// TwinCAT 3 PLC project PLC
// ProgramVersion: 3.1.4023.0
// libraries:
//   Tc2_Standard, * (Beckhoff Automation GmbH)
//   Tc2_System, * (Beckhoff Automation GmbH)
//   Tc3_Module, * (Beckhoff Automation GmbH)
//   VisuDialogs, * (System)
//   VisuSymbols,3.5.10.0,System
// project tree:
//   / GlobalTextList.TcGTLO, PlcTask.TcTTO, Visualization Manager.TcVMO (not stored)
//   POUs/ FB_Blinker.TcPOU, MAIN.TcPOU, pCounter.TcPOU
//   VISUs/ P03_Common.TcVIS, P00_Main.TcVIS, P02_Measurement.TcVIS, P01_Swtich_Lamp.TcVIS, P04_Table.TcVIS, TextList.TcTLO, W01_PopupScreen.TcVIS

CONFIGURATION PLC
    RESOURCE PLC ON TwinCAT3
        TASK PlcTask(INTERVAL := T#10ms, PRIORITY := 20);
        PROGRAM MAIN WITH PlcTask : MAIN;
    END_RESOURCE
END_CONFIGURATION

// ---- POUs/MAIN.TcPOU
PROGRAM MAIN
VAR 	
	bHmi_LAMP1  : BOOL;
	bHmi_LAMP2 : BOOL;
	bHmi_LAMP3  : BOOL;
	bHmi_LAMP4  : BOOL;
	
//	bOut_LAMP1  AT %Q*: BOOL;
//	bOut_LAMP2  AT %Q*: BOOL;
//	bOut_LAMP3  AT %Q*: BOOL;
//	bOut_LAMP4  AT %Q*: BOOL;
	
	bHmi_Swtic1 : BOOL;
	bHmi_Swtic2 : BOOL;
	bHmi_Swtic3 : BOOL;
	bHmi_Swtic4 : BOOL;
	
//	bIn_Swtic1 AT %I*: BOOL;
//	bIn_Swtic2 AT %I*: BOOL;
//	bIn_Swtic3 AT %I*: BOOL;
//	bIn_Swtic4 AT %I*: BOOL;
	
	iIN_VOLUME AT %I*: INT:=1000;
	
	//bIN_SW2 AT %I*: BOOL;
	fbBlinker: FB_Blinker;
	fbCTU: CTU;
	
	//HMI  BarDisplay
	iValueBarDisplay:INT;
	tTimer:TON;
	bDirection:BOOL;
	bValuePotentialMeter:INT;
	
	//Bar Graph
	lrSin:LREAL;
	aryLrSin:ARRAY[0..200] OF LREAL;
	tTimer2:TON;
	i:INT;
	
	//check Box
	bCheckBox:ARRAY[0..4] OF BOOL;
	bCheckBox1:BOOL;
	bCheckBox2:BOOL;
	bCheckBox3:BOOL;
	bCheckBox4:BOOL;
	bCheckBox5:BOOL;
	plsCheckBox1:R_trig;
	plsCheckBox2:R_trig;
	plsCheckBox3:R_trig;
	plsCheckBox4:R_trig;
	plsCheckBox5:R_trig;
	sOutput2:STRING;
	//Combbox and Radio Buttons
	iCombINdex:INT;
	sOutput:STRING;
	
    //Table 
	aryLrSin1:ARRAY[0..4,0..20] OF DINT;
	tTimer3:TON;
END_VAR

//bOUT_LAMP1:=bIN_SW1;
//iOUT_METER:=iIN_VOLUME;
//bOUT_LAMP3:= bIN_SW1 AND bIN_SW2;

//pCounter();

fbBlinker
(
//	bStart:=TRUE,
	bStart:=bHmi_Swtic1,
	tTime:=INT_TO_TIME(iIN_VOLUME),
	//bOutPut=>
);

fbCTU(
	CU:= fbBlinker.bOutPut, 
	RESET:= fbCTU.Q, 
	PV:= 4, 
	//Q=> , 
	//CV=> 
);

CASE fbCTU.CV OF 
	1: 
	bHmi_LAMP1:=TRUE;
	bHmi_LAMP2:=FALSE;
	bHmi_LAMP3:=FALSE;
	bHmi_LAMP4:=FALSE;
	2: 
	bHmi_LAMP1:=FALSE;
	bHmi_LAMP2:=TRUE;
	bHmi_LAMP3:=FALSE;
	bHmi_LAMP4:=FALSE;
	3: 
	bHmi_LAMP1:=FALSE;
	bHmi_LAMP2:=FALSE;
	bHmi_LAMP3:=TRUE;
	bHmi_LAMP4:=FALSE;
	4: 
	bHmi_LAMP1:=FALSE;
	bHmi_LAMP2:=FALSE;
	bHmi_LAMP3:=FALSE;
	bHmi_LAMP4:=TRUE;

END_CASE

//Hmi BarDisplay
tTimer(IN:=bHmi_Swtic2,PT:=T#10MS);
IF tTimer.Q THEN
	tTimer(IN:=FALSE);
	IF iValueBarDisplay = 1000 THEN
		bDirection:=TRUE;
	ELSIF iValueBarDisplay = 0 THEN
		bDirection:=FALSE;	
	END_IF
	
	IF bDirection THEN
		iValueBarDisplay:=iValueBarDisplay-1;
	ELSE
		iValueBarDisplay:=iValueBarDisplay+1;
	END_IF
END_IF

//HMI Bar Graph
lrSin:=SIN(TO_REAL(iValueBarDisplay)/1000);
tTimer2(IN:=bHmi_Swtic3,PT:=T#100MS);
IF tTimer2.Q THEN
	tTimer2(IN:=FALSE);
	FOR i:= 200 TO 1 BY -1 DO 
		aryLrSin[i]:=aryLrSin[i-1];
	END_FOR
	aryLrSin[0]:=LrSin;
END_IF
//CheckBox
plsCheckBox1(CLK:=bCheckBox1);
plsCheckBox2(CLK:=bCheckBox2);
plsCheckBox3(CLK:=bCheckBox3);
plsCheckBox4(CLK:=bCheckBox4);
plsCheckBox5(CLK:=bCheckBox5);
IF plsCheckBox1.Q THEN
	sOutput2:='Opton1';
	bCheckBox2:=FALSE;	
	bCheckBox3:=FALSE;	
	bCheckBox4:=FALSE;	
	bCheckBox5:=FALSE;	
ELSIF plsCheckBox2.Q THEN
	sOutput2:='Opton2';
	bCheckBox1:=FALSE;	
	bCheckBox3:=FALSE;	
	bCheckBox4:=FALSE;	
	bCheckBox5:=FALSE;	
ELSIF plsCheckBox3.Q THEN
	sOutput2:='Opton3';
	bCheckBox1:=FALSE;	
	bCheckBox2:=FALSE;	
	bCheckBox4:=FALSE;	
	bCheckBox5:=FALSE;		
ELSIF plsCheckBox4.Q THEN
	sOutput2:='Opton4';
	bCheckBox1:=FALSE;	
	bCheckBox2:=FALSE;	
	bCheckBox3:=FALSE;	
	bCheckBox5:=FALSE;	
ELSIF plsCheckBox5.Q THEN
	sOutput2:='Opton5';
	bCheckBox1:=FALSE;	
	bCheckBox2:=FALSE;	
	bCheckBox3:=FALSE;	
	bCheckBox4:=FALSE;	
END_IF
//CombBox
CASE iCombINdex OF
0:
 sOutput:='Opton1';
1:
 sOutput:='Opton2';
2:
 sOutput:='Opton3';
3:
 sOutput:='Opton4';
ELSE
 sOutput:='Error';
END_CASE
//Table
tTimer3(IN:=bHmi_Swtic4,PT:=T#1000MS);
IF tTimer3.Q THEN
	tTimer3(IN:=FALSE);
	FOR i:= 20 TO 1 BY -1 DO 
		aryLrSin1[0,i]:=aryLrSin1[0,i-1];
		aryLrSin1[1,i]:=aryLrSin1[1,i-1];
		aryLrSin1[2,i]:=aryLrSin1[2,i-1];
		aryLrSin1[3,i]:=aryLrSin1[3,i-1];
		aryLrSin1[4,i]:=aryLrSin1[4,i-1];
	END_FOR
	aryLrSin1[0,0]:=TO_DINT(LrSin*10000);
	aryLrSin1[1,0]:=TO_DINT(-LrSin*10000);
	aryLrSin1[2,0]:=TO_DINT((LrSin+1)*10000);
	aryLrSin1[3,0]:=TO_DINT((LrSin-1)*10000);
	aryLrSin1[4,0]:=TO_DINT((LrSin*2)*10000);
END_IF

END_PROGRAM

// ---- POUs/FB_Blinker.TcPOU
FUNCTION_BLOCK FB_Blinker
VAR_INPUT
	bStart: BOOL;
	tTime: TIME;
END_VAR
VAR_OUTPUT
	bOutPut: BOOL;
END_VAR
VAR
	T1: TON;
	T2: TON;
END_VAR

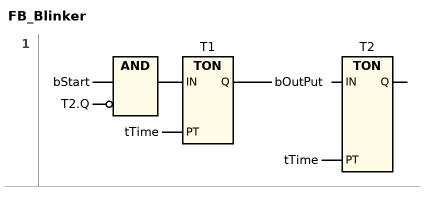
// NETWORK 1
T1(IN := bStart AND NOT T2.Q, PT := tTime); // TON
bOutPut := T1.Q;
T2(IN := T1.Q, PT := tTime); // TON

END_FUNCTION_BLOCK

// ---- POUs/pCounter.TcPOU
PROGRAM pCounter
VAR
	fbCTU: CTU;
	bSW1 AT %I*: BOOL;
	bSW2 AT %I*: BOOL;
	CurrentValue: WORD;
	bLED1 AT %Q*: BOOL;
END_VAR

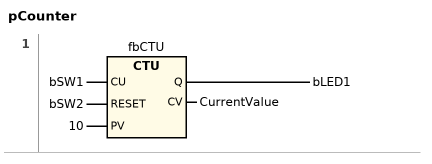
// NETWORK 1
fbCTU(CU := bSW1, RESET := bSW2, PV := 10, CV => CurrentValue); // CTU
bLED1 := fbCTU.Q;

END_PROGRAM

// ---- GlobalTextList.TcGTLO
TEXTLIST GlobalTextList
  646 = '%d'
  394 = '%s'
  322 = 'aryLrSiin1[1]'
  243 = 'aryLrSin1[0,INDEX]'
  253 = 'aryLrSin1[0]'
  589 = 'aryLrSin1[1,INDEX]'
  141 = 'aryLrSin1[1]'
  425 = 'aryLrSin1[2,INDEX]'
  682 = 'aryLrSin1[2]'
  644 = 'aryLrSin1[3,INDEX]'
  914 = 'aryLrSin1[3]'
  670 = 'aryLrSin1[4,INDEX]'
  300 = 'aryLrSin1[4]'
  706 = 'aryLrSin1[X]'
  594 = 'Bar_Switch_2'
  122 = 'Chart_Switch_3'
  446 = 'Check Box'
  607 = 'Check Box1'
  567 = 'Checkbox'
  756 = 'CheckBox'
  353 = 'Checkbox1'
  536 = 'Checkbox2'
  535 = 'Checkbox3'
  854 = 'Close Screen'
  739 = 'Close Window'
  413 = 'Common'
  320 = 'GroupBox'
  554 = 'Here PopUp\u3000'
  537 = 'Here PopUp\u3000TEXT\u3000'
  943 = 'Japanese'
  485 = 'Lamp_1' | JP: 'ランプ１'
  549 = 'Lamp_2' | JP: 'ランプ２'
  964 = 'Lamp_3' | JP: 'ランプ３'
  83 = 'Lamp_4' | JP: 'ランプ４'
  254 = 'Lamp_Switch_1'
  906 = 'Measument'
  348 = 'Measurement'
  331 = 'OpenPopup'
  733 = 'Option1'
  643 = 'Option14'
  808 = 'Option2'
  403 = 'Option3'
  186 = 'Option4'
  115 = 'Option5'
  754 = 'PopUp Window'
  588 = 'Switch 1'
  163 = 'Switch 2'
  482 = 'Switch 3'
  888 = 'Switch 4'
  357 = 'Switch Time' | JP: 'スイッチ時間'
  496 = 'Switch Time Act' | JP: '実時間'
  905 = 'Switch_1' | JP: 'スイッチ１'
  363 = 'Switch_2' | JP: 'スイッチ２'
  119 = 'Switch_3' | JP: 'スイッチ３'
  130 = 'Switch_4' | JP: 'スイッチ４'
  404 = 'swtich Lamp'
  929 = 'Swtich Time'
  542 = 'Table'
  559 = 'Table_Switch_4'
END_TEXTLIST

// ---- VISUs/P03_Common.TcVIS
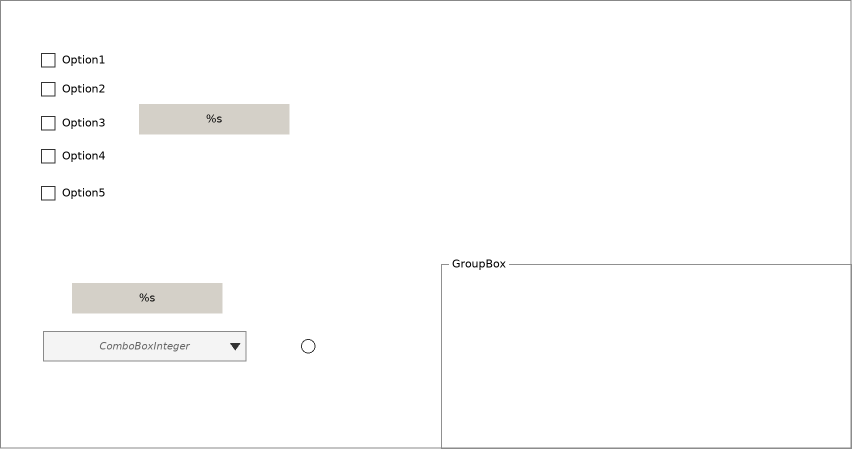
VISUALIZATION P03_Common  // 852x449
    Checkbox (39,45 150x30), "Option1", variable: Main.bCheckBox1
    Checkbox (39,74 150x30), "Option2", variable: Main.bCheckBox2
    Checkbox (39,108 150x30), "Option3", variable: Main.bCheckBox3
    Checkbox (39,141 150x30), "Option4", variable: Main.bCheckBox4
    Checkbox (39,178 150x30), "Option5", variable: Main.bCheckBox5
    Textfield (139,104 150x30), "%s", text variable: Main.sOutput2
    ComboBoxInteger (43,331 203x30), variable: Main.iCombINdex, text list: 'TextList'
    RadioButton (299,271 150x150), variable: Main.iCombINdex
        Areas[0]: Text=Option1
        Areas[1]: Text=Option2
        Areas[2]: Text=Option3
        Areas[3]: Text=Option4
        Areas[4]: Text=Option5
    Textfield (72,283 150x30), "%s", text variable: Main.sOutput
    GroupBox (441,256 411x193), "GroupBox"
END_VISUALIZATION

// ---- VISUs/P00_Main.TcVIS
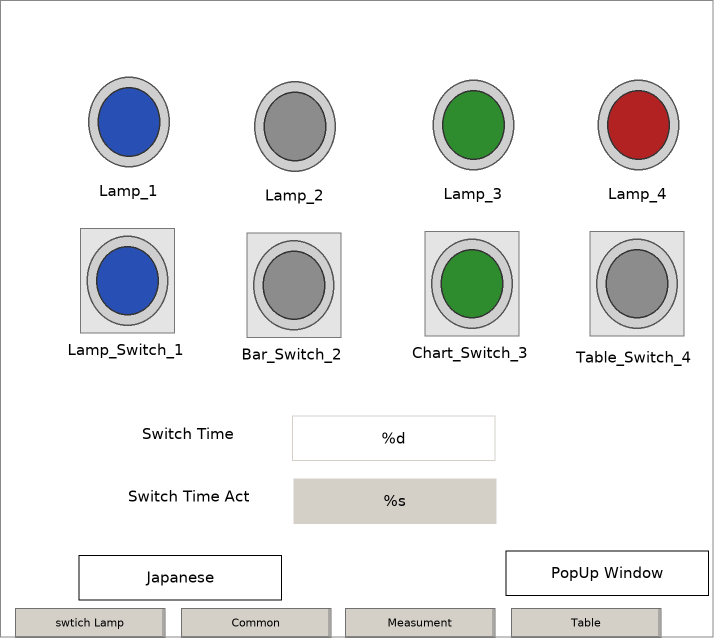
VISUALIZATION P00_Main  // 714x638
    Button (15,608 150x30), "swtich Lamp"
        OnMouseDown: FrameSelectionChange Selection=SelectedFrame=647e187a-0755-4409-bbed-ce6851db0410, GlobSel=AssignType=Directly, SelType=Locally
    Frame (29,26 685x574)
        shows P01_Swtich_Lamp()
        shows P02_Measurement()
        shows P03_Common()
        shows P04_Table()
    Button (181,608 150x30), "Common"
        OnMouseDown: FrameSelectionChange Selection=SelectedFrame=647e187a-0755-4409-bbed-ce6851db0410, Selection=2, GlobSel=AssignType=Directly, SelType=Locally
    Button (345,608 150x30), "Measument"
        OnMouseDown: FrameSelectionChange Selection=SelectedFrame=647e187a-0755-4409-bbed-ce6851db0410, Selection=1, GlobSel=AssignType=Directly, SelType=Locally
    Button (511,608 150x30), "Table"
        OnMouseDown: FrameSelectionChange Selection=SelectedFrame=647e187a-0755-4409-bbed-ce6851db0410, Selection=3, GlobSel=AssignType=Directly, SelType=Locally
END_VISUALIZATION

// ---- VISUs/P02_Measurement.TcVIS
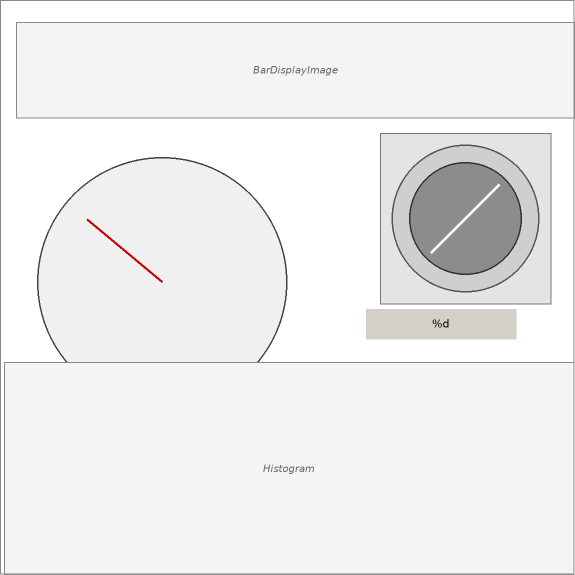
VISUALIZATION P02_Measurement  // 575x575
    BarDisplayImage (16,22 559x96), value: Main.iValueBarDisplay, style: BarDisplayImage-Gray, scale format: %.1f, scale 0..1000
    Meter180 (37,157 250x250), value: Main.iValueBarDisplay, style: Meter-Meter180-Gray, scale format: %.1f, scale 0..1000
    Potentiometer360 (362,133 207x171), variable: Main.bValuePotentialMeter, style: Potentiometer-Potentiometer360-Gray, scale format: %.1f, scale 0..100
        p2431819421: Outside
    Textfield (366,309 150x30), "%d", text variable: Main.bValuePotentialMeter
    Histogram (4,362 570x213), scale format: %.1f, scale 0..1
        p1518820177: Main.aryLrSin
        p102497268: Main.aryLrSin
        p788070771: ARRAY [0..200] OF LREAL
END_VISUALIZATION

// ---- VISUs/P01_Swtich_Lamp.TcVIS
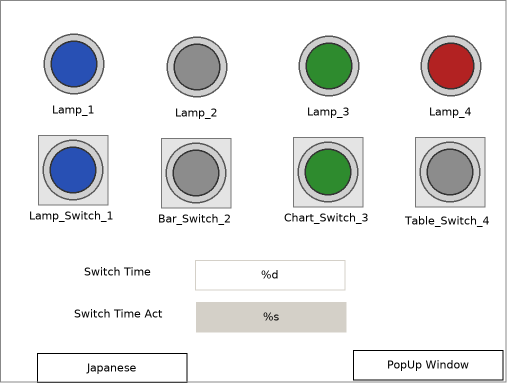
VISUALIZATION P01_Swtich_Lamp  // 507x383
    Lamp1 (39,29 70x70), variable: Main.bHmi_LAMP1, style: Lamp-Lamp1-Blue
    Label (17,95 113x30), "Lamp_1"
    PushSwitch (38,135 70x70), variable: Main.bHmi_Swtic1, behaviour: TOGGLE, style: Switch-PushSwitch-Blue
    Label (15,201 113x30), "Lamp_Switch_1"
    Lamp1 (162,32 70x70), variable: Main.bHmi_LAMP2, style: Lamp-Lamp1-Gray
    Label (140,98 113x30), "Lamp_2"
    PushSwitch (161,138 70x70), variable: Main.bHmi_Swtic2, behaviour: TOGGLE, style: Switch-PushSwitch-Gray
    Label (138,204 113x30), "Bar_Switch_2"
    Lamp1 (294,31 70x70), variable: Main.bHmi_LAMP3, style: Lamp-Lamp1-Green
    Label (272,97 113x30), "Lamp_3"
    PushSwitch (293,137 70x70), variable: Main.bHmi_Swtic3, behaviour: TOGGLE, style: Switch-PushSwitch-Green
    Label (270,203 113x30), "Chart_Switch_3"
    Lamp1 (416,31 70x70), variable: Main.bHmi_LAMP4, style: Lamp-Lamp1-Red
    Label (394,97 113x30), "Lamp_4"
    PushSwitch (415,137 70x70), variable: Main.bHmi_Swtic4, behaviour: TOGGLE, style: Switch-PushSwitch-Gray
    Label (391,206 113x30), "Table_Switch_4"
    Textfield (195,260 150x30), "%d", text variable: Main.iIN_VOLUME
        OnMouseUp: write the text variable via Default
    Label (61,257 113x30), "Switch Time"
    Textfield (196,302 150x30), "%s", text variable: MAIN.fbBlinker.T1.ET
    Label (62,299 113x30), "Switch Time Act"
    RoundedRectangle (37,353 150x30), "Japanese"
        OnMouseClick: ChangeLanguage ChangeLanguage=JP
    RoundedRectangle (353,350 150x30), "PopUp Window"
        OnMouseClick: OpenDialog Dialog=W01_PopupScreen, OpenModal=True, OpenCentered=True
END_VISUALIZATION

// ---- VISUs/P04_Table.TcVIS
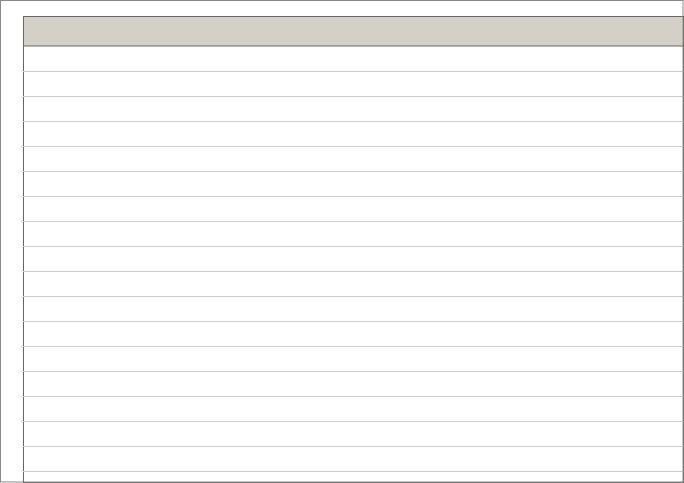
VISUALIZATION P04_Table  // 684x483
    Table (23,16 661x467), data array: Main.aryLrSin1
        p3854506369: Main.aryLrSin1[0,INDEX]
        p1892666644: Main.aryLrSin1[1,INDEX]
        p338671338: Main.aryLrSin1[2,INDEX]
        p2170511999: Main.aryLrSin1[3,INDEX]
        p3723444502: Main.aryLrSin1[4,INDEX]
        p2232123230: aryLrSin1[0]
        p511219082: aryLrSiin1[1]
        p1755163831: aryLrSin1[2]
        p4092479075: aryLrSin1[3]
        p2237128397: aryLrSin1[4]
END_VISUALIZATION

// ---- VISUs/TextList.TcTLO
TEXTLIST TextList
  0 = 'Option1'
  1 = 'Option2'
  2 = 'Option3'
  3 = 'Option4'
  4 = 'Option5'
   = ''
END_TEXTLIST

// ---- VISUs/W01_PopupScreen.TcVIS
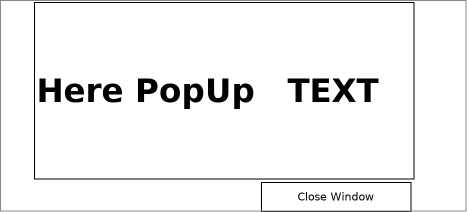
VISUALIZATION W01_PopupScreen  // 467x212
    Label (24,34 443x139)
    RoundedRectangle (261,182 150x30), "Close Window"
        OnMouseClick: CloseDialog Dialog=W01_PopupScreen, Result=OK, NumpadKeypadSet=True
    Rectangle (34,2 380x177), "Here PopUp TEXT"
END_VISUALIZATION
